// Mitsubishi GX Works2 project: Texto Estruturado   PLC: Q03UDV

// task Task_01 (event TRUE, interval 0, priority 31): POU_01
// task stteste (event TRUE, interval 0, priority 31): stteste

PROGRAM POU_01
VAR
  iDR : ARRAY [0..4] OF INT;
END_VAR
VAR CONSTANT
  iElement2 : INT := 4;
  iElemet1 : INT := 9;
END_VAR
iDR[0] := iElemet1 + iElement2 ;
iDR[1] := iElemet1 - iElement2 ; 
iDR[2] := iElemet1 * iElement2 ; 
(*Codesys*)
iDR[3] := iElemet1 / iElement2 ; 
iDR[4] := iElemet1 MOD iElement2;
END_PROGRAM

FUNCTION fSoma
VAR_INPUT
  iEle1 : INT;
  iEle2 : INT;
END_VAR
fSoma := iEle1 + iEle2;
END_FUNCTION

PROGRAM stteste
VAR
  iLeo : INT;
END_VAR
iLeo := fSoma( 100 , 450 );
END_PROGRAM
